// TwinCAT 3 PLC project PLC_FIS
// ProgramVersion: 3.1.4024.12
// libraries:
//   Tc2_Standard, * (Beckhoff Automation GmbH)
//   Tc2_System, * (Beckhoff Automation GmbH)
//   Tc3_Module, * (Beckhoff Automation GmbH)
// project tree:
//   UserDefinedTypes/ eAndMethod.TcDUT (not stored), eDeffuzyMethod.TcDUT, eOrMethod.TcDUT, eTest.TcDUT (not stored), MAMFIS.TcDUT (not stored), FIS_RULES.TcDUT (not stored), FIS_VAR.TcDUT (not stored), FIS_VAR_1.TcDUT, MF_INDEX.TcDUT (not stored), MF_SHAPE.TcDUT (not stored), MEMBERSHIP_FUNCTION.TcDUT
//   GlobalVariables/ gvlFIS_Constants.TcGVL (not stored)
//   / PlcTask.TcTTO
//   FUNS_and_FB/Deffuzzification/ fCentroid.TcPOU
//   FUNS_and_FB/ FB_AGGREGATION.TcPOU, FB_IMPLICATION.TcPOU
//   FUNS_and_FB/Fuzzification/ fMembershipDegree.TcPOU (not stored), fMembershipDegreeArray.TcPOU (not stored)
//   FUNS_and_FB/Fuzzification/Membership Functions/ MF_Gaussian.TcPOU (not stored), MF_L.TcPOU (not stored), MF_R.TcPOU (not stored), MF_S.TcPOU, MF_Sigmoidal.TcPOU (not stored), MF_Singleton.TcPOU (not stored), MF_Trapezoidal.TcPOU, MF_Triangular.TcPOU (not stored), MF_Z.TcPOU (not stored)
//   FUNS_and_FB/FuzzyOperations/ fuzzyset.TcPOU (not stored), FuzzyAND_array.TcPOU, fuzzyAND.TcPOU (not stored), FuzzyNOT.TcPOU (not stored), FuzzyOR_array.TcPOU, FuzzyOR.TcPOU (not stored)
//   FUNS_and_FB/FuzzyOperations/T-Norms/ TN_min.TcPOU, TN_prod.TcPOU (not stored)
//   FUNS_and_FB/_FuzzyInferenceSystem/ FB_FIS_MAMDANI.TcPOU (not stored)
//   _Main/ MAIN.TcPOU, Test_fbFis.TcPOU

CONFIGURATION PLC_FIS
    RESOURCE PLC ON TwinCAT3
        TASK PlcTask(INTERVAL := T#1ms, PRIORITY := 20);
        PROGRAM MAIN WITH PlcTask : MAIN;
    END_RESOURCE
END_CONFIGURATION

// ---- UserDefinedTypes/eDeffuzyMethod.TcDUT
//{attribute 'qualified_only'}
{attribute 'strict'}
TYPE eDeffuzyMethod :
(
	Centroid
);
END_TYPE

// ---- UserDefinedTypes/eOrMethod.TcDUT
//{attribute 'qualified_only'}
{attribute 'strict'}
TYPE eOrMethod :
(
	Maximum
);
END_TYPE

// ---- UserDefinedTypes/FIS_VAR_1.TcDUT
TYPE FIS_VAR_1 :
STRUCT
	Signal:  REAL;
	//MyVarInfo :__SYSTEM.VAR_INFO:=__VARINFO(Signal);
	//Name:STRING:=MyVarInfo.Symbol;
	Range:ARRAY[0..1] OF REAL;
	NumberOfMF:INT;
	MF:ARRAY [1..9]OF MEMBERSHIP_FUNCTION;
	
END_STRUCT
END_TYPE

// ---- UserDefinedTypes/MEMBERSHIP_FUNCTION.TcDUT
TYPE MEMBERSHIP_FUNCTION :
	STRUCT
		Name:STRING;
		Shape: MF_SHAPE;//membership function shape
		//MfPoints: ARRAY[*]OF REAL;//membership funciton points
		Points: ARRAY[1..5]OF REAL;
	END_STRUCT
END_TYPE

// ---- _Main/MAIN.TcPOU
PROGRAM MAIN
VAR
END_VAR

Test_fbFis();

END_PROGRAM

// ---- _Main/Test_fbFis.TcPOU
PROGRAM Test_fbFis
VAR
	Input1Simulation,Input2Simulation,OutputSimulation: REAL;
	fbFIS:FB_FIS_MAMDANI;
	FIS:MAMFIS;
END_VAR

//FIS parameters========================================
FIS.Name:='LaserHeatControl2';

//FIS.Inputs DEFINITION=================================
	//input1=ERROR(command-feedback)
		FIS.Inputs[Error].CrispValue:=	Input1Simulation;
		FIS.Inputs[Error].Name  :=  	'TempError';
		FIS.Inputs[Error].Range[1] :=  	0;
		FIS.Inputs[Error].Range[2] := 	70;
		FIS.Inputs[Error].NumberOfMF := 3;
		//MF NONE
			FIS.Inputs[1].MF[1].Name := 	'none';
			FIS.Inputs[1].MF[1].Shape := 	MF_SHAPE.Rshaped;
			FIS.Inputs[1].MF[1].Points[1] := 0;
			FIS.Inputs[1].MF[1].Points[2] := 10;
		//MF LITTLE	
			FIS.Inputs[1].MF[2].Name := 	'litle';
			FIS.Inputs[1].MF[2].Shape := 	MF_SHAPE.Triangular;
			FIS.Inputs[1].MF[2].Points[1] := 5;
			FIS.Inputs[1].MF[2].Points[2] := 20;
			FIS.Inputs[1].MF[2].Points[3] := 40;
		//MF BIG	
			FIS.Inputs[1].MF[3].Name := 	'big';                                                                                 
			FIS.Inputs[1].MF[3].Shape := 	MF_SHAPE.Lshaped;
			FIS.Inputs[1].MF[3].Points[1] := 20;
			FIS.Inputs[1].MF[3].Points[2] := 60;	
											 
	//input2=SPEED
		FIS.Inputs[2].CrispValue:=	Input2Simulation;
		FIS.Inputs[2].Name := 		'speed';
		FIS.Inputs[2].Range[1] :=  	0;
		FIS.Inputs[2].Range[2] := 	20;
		FIS.Inputs[2].NumberOfMF := 3;
		
		FIS.Inputs[2].MF[1].Name := 	'null';
		FIS.Inputs[2].MF[1].Shape := 	MF_SHAPE.Rshaped;
		FIS.Inputs[2].MF[1].Points[1] := 0;
		FIS.Inputs[2].MF[1].Points[2] := 2;
		
		FIS.Inputs[2].MF[2].Name := 	'litlle';
		FIS.Inputs[2].MF[2].Shape := 	MF_SHAPE.Triangular;
		FIS.Inputs[2].MF[2].Points[1] := 0;
		FIS.Inputs[2].MF[2].Points[2] := 5;
		FIS.Inputs[2].MF[2].Points[3] := 10;
		
		FIS.Inputs[2].MF[3].Name := 	'Big';
		FIS.Inputs[2].MF[3].Shape := 	MF_SHAPE.Lshaped;
		FIS.Inputs[2].MF[3].Points[1] := 8;
		FIS.Inputs[2].MF[3].Points[2] := 15;
//======================================================

//FUZZY FIS.Outputs DEFINITION =========================
	FIS.Outputs[1].Name  :=  		'Power';
	FIS.Outputs[1].Range[1] :=  	0;
	FIS.Outputs[1].Range[2] :=		120;
	FIS.Outputs[1].NumberOfMF := 	3;
	//MF LOW
		FIS.Outputs[1].MF[1].Name := 	'Low';
		FIS.Outputs[1].MF[1].Shape := 	MF_SHAPE.Rshaped;
		FIS.Outputs[1].MF[1].Points[1] := 0;
		FIS.Outputs[1].MF[1].Points[2] := 30 ;
	//MF MEDIUM
		FIS.Outputs[Power].MF[Medium].Name := 	'Medium';
		FIS.Outputs[Power].MF[Medium].Shape := 	MF_SHAPE.Triangular;
		FIS.Outputs[Power].MF[Medium].Points[1] := 20;
		FIS.Outputs[Power].MF[Medium].Points[2] := 40;
		FIS.Outputs[Power].MF[Medium].Points[3] := 60;
	//MF HIGH	
		FIS.Outputs[Power].MF[High].Name := 'High';
		FIS.Outputs[Power].MF[High].Shape := MF_SHAPE.Lshaped;
		FIS.Outputs[Power].MF[High].Points[1] := 50;
		FIS.Outputs[Power].MF[High].Points[2] := 100;
//======================================================

//FUZZY_rules===========================================
	//Rule 1
		FIS.Rules[1].Antecedent := FIS.MD[error,none];
		FIS.Rules[1].Consequents[power] := low;
	//Rule 2
		FIS.Rules[2].Antecedent:=FIS.MD[error,little];
		FIS.Rules[2].Consequents[power] := medium;
	//Rule 3
		FIS.Rules[3].Antecedent:= FIS.MD[error,big];
		FIS.Rules[3].Consequents[power] := High;
//======================================================
//FIS INSTANTIATION========================================
fbFIS(FIS:=FIS);
OutputSimulation:=fis.Outputs[1].CrispValue;

END_PROGRAM

// ---- FUNS_and_FB/Deffuzzification/fCentroid.TcPOU
FUNCTION fCentroid : REAL
VAR_INPUT
	resolution:DINT;//number of integration rectangles
	Range:ARRAY[1..2] OF REAL;
	fbAggregation: REFERENCE TO FB_AGGREGATION;//MF:MEMBERSHIP_FUNCTION;
END_VAR
VAR
	i:DINT;
	Xi,MDi:REAL;
	IntegrationStep: REAL;
	Dividend:REAL:=0;//sum(MD(Xi))
 	Divisor:REAL:=0;//sum(Xi*MD(Xi))
END_VAR
VAR_OUTPUT
	error:BOOL:=FALSE;
END_VAR

(*
centroid=   sum(Xi*MD(Xi))  dividend
		   ===============
		     sum(MD(Xi)) divisor
*)
IF Resolution<>0 THEN
	IntegrationStep :=(Range[2]-Range[1])/DINT_TO_REAL(Resolution);
	FOR i := 1 TO resolution DO
		Xi := DINT_TO_REAL(i)*IntegrationStep;
		fbAggregation(X:=Xi);
		MDi := fbAggregation.FSValue;
		Dividend := Dividend +Xi* MDi*IntegrationStep;
		Divisor := Divisor + MDi*IntegrationStep;
	END_FOR
	IF Divisor<>0 THEN
		fCentroid := Dividend/Divisor;
	ELSE
		fCentroid:=0;
	END_IF
ELSE error:=TRUE;	
END_IF

END_FUNCTION

// ---- FUNS_and_FB/FB_AGGREGATION.TcPOU
FUNCTION_BLOCK FB_AGGREGATION
VAR_INPUT
	//fbImplication: REFERENCE TO FB_IMPLICATION;
	Myrules:ARRAY [1..NumOfFisRules] OF FIS_RULES;
	MyFISoutputs:ARRAY [1..NumOfFISOutputs] OF FIS_VAR;
	X:REAL;
END_VAR

VAR
	firstRule,LastRule,i,j:DINT;
	aofFuzzySet:  ARRAY [1..NumOfFisRules] OF REAL;
	fbImplication:FB_IMPLICATION;
	MyMF: INT;
END_VAR
VAR_OUTPUT
	FSValue:REAL; 
END_VAR

//firstRule:=LOWER_BOUND(Rule,1);
//LastRule:=UPPER_BOUND(Rule,1);
//FOR i:=firstRule TO LastRule DO
FOR i:=1 TO NumOfFisRules DO
	FOR j:=1 TO NumOfFISOutputs DO
		IF Myrules[i].Consequents[j]>0 THEN
		MyMF:=Myrules[i].Consequents[j];
		fbImplication(
				X:=X,
				Antecedent:=Myrules[i].Antecedent,
				FISOutputMf:= MyFISoutputs[j].MF[MyMF]);
		aofFuzzySet[i]:=fbImplication.RuleFuzzySet;
		END_IF
	END_FOR
END_FOR

FSValue:=FuzzyOR_array(maximum,aofFuzzySet);

END_FUNCTION_BLOCK

// ---- FUNS_and_FB/FB_IMPLICATION.TcPOU
FUNCTION_BLOCK FB_IMPLICATION
VAR_INPUT
	Antecedent: REAL;
	X:REAL;
	FISOutputMf: MEMBERSHIP_FUNCTION;
END_VAR
VAR_OUTPUT
	RuleFuzzySet:REAL;
END_VAR

RuleFuzzySet :=fuzzyAND(Minimum,fMembershipDegree(x,FISOutputMf),Antecedent);

END_FUNCTION_BLOCK

// ---- FUNS_and_FB/FuzzyOperations/FuzzyOR_array.TcPOU
FUNCTION FuzzyOR_array : real
VAR_INPUT
	ORmethod:eOrMethod;
END_VAR
VAR_IN_OUT
	Inputs:ARRAY[*]OF REAL;
END_VAR

VAR
	i: DINT;
END_VAR

FuzzyOR_array:=0;
FOR i:=LOWER_BOUND(Inputs,1) TO UPPER_BOUND(Inputs,1) DO
	IF inputs[i] > FuzzyOR_array THEN
		FuzzyOR_array := inputs[i];
	END_IF
END_FOR

END_FUNCTION

// ---- FUNS_and_FB/Fuzzification/Membership Functions/MF_S.TcPOU
FUNCTION MF_S : real
VAR_INPUT
	x,a,b:REAL;(*a defines the foot of the membership function, AND b defines its shoulder.*)

END_VAR
VAR_OUTPUT
	Error:BOOL;
END_VAR

IF NOT(b=a) THEN
	IF x<=a THEN
		MF_S := 0;
	ELSIF a<=x AND x<=(a+b)/2 THEN
		MF_S := LREAL_TO_REAL( 2*EXPT(((x-a)/(b-a)),2));
	ELSIF (a+b)/2<=x AND x<=b THEN
		MF_S := 1 - 2*LREAL_TO_REAL(EXPT(((x-b)/(b-a)),2));
	ELSIF b<=x THEN
		MF_S := 1;
	END_IF
ELSE
	Error:=TRUE;
END_IF

END_FUNCTION

// ---- FUNS_and_FB/Fuzzification/Membership Functions/MF_Trapezoidal.TcPOU
FUNCTION MF_Trapezoidal : real
VAR_INPUT
	x,a,b,c,d:REAL;
END_VAR
VAR_OUTPUT
	Error:BOOL;
END_VAR

//a < b < c < d
IF NOT(b=a OR d=c) AND
(a<b) AND (b<c) AND (c<d) THEN
	IF x<a THEN
		MF_Trapezoidal:=0;
	ELSIF a<=x AND x<=b THEN
		MF_Trapezoidal:=(x-a)/(b-a);
	ELSIF b<=x AND x<=c THEN
		MF_Trapezoidal:=1;
	ELSIF d<=x AND x<=c THEN
		MF_Trapezoidal:=(d-x)/(d-c);
	END_IF
ELSE
	Error:=TRUE;		
END_IF

END_FUNCTION

// ---- FUNS_and_FB/FuzzyOperations/FuzzyAND_array.TcPOU
FUNCTION FuzzyAND_array : real
VAR_INPUT
	ANDmethod:eAndMethod;
END_VAR
VAR_IN_OUT
	Inputs:ARRAY[*]OF REAL;
END_VAR

CASE ANDmethod OF
	eAndMethod.Minimum://***********
		FuzzyAND_array := TN_min(Inputs);
	eAndMethod.Product://***********
		FuzzyAND_array := TN_prod(Inputs);
END_CASE

END_FUNCTION

// ---- FUNS_and_FB/FuzzyOperations/T-Norms/TN_min.TcPOU
FUNCTION TN_min : real
VAR
	i:DINT;
END_VAR
VAR_IN_OUT
	Inputs: ARRAY[*] OF REAL;
END_VAR

FOR i:=LOWER_BOUND(Inputs,1) TO UPPER_BOUND(Inputs,1) DO
	IF inputs[i] < TN_min THEN
		TN_min:=inputs[i];
	END_IF
END_FOR

END_FUNCTION
